{attribute 'qualified_only'}
{attribute 'strict'}
TYPE E_Base :
(
	{attribute 'hide'} 
	Init 	:= 0,
	Starting:= 2,	
	Execute	:= 3,
	Stopping:= 4,
	Aborting:= 5,
	Aborted	:= 6,
	Reset	:= 7,
	Stopped	:= 1
)USINT;
END_TYPE

(* stored: Version 1.1.0.1
   DUT E_Base: Id {a98106f4-9ac5-049b-0182-44b4aa9fecc7} *)
